FUNCTION_BLOCK FB_GenerateHeartBeat
VAR_INPUT
END_VAR
VAR_OUTPUT
	iHeartBeat		: UINT;
END_VAR
VAR
	tInterval		: TIME := T#500ms;
	tonInterval		: TON;
END_VAR


tonInterval(IN := TRUE,
			PT := tInterval,
			Q => );

IF (tonInterval.Q) THEN
	tonInterval(IN := FALSE);
	iHeartBeat := iHeartBeat + 1;
	IF (iHeartBeat > 100) THEN
		iHeartBeat := 0;
	END_IF
END_IF

PROPERTY PUBLIC P_tInterval : TIME
GET
P_tInterval := tInterval;
END_GET
SET
tInterval := P_tInterval;
END_SET
END_PROPERTY

END_FUNCTION_BLOCK

(* stored: Version 1.1.0.1, ProductVersion 3.1.4024.2
   POU FB_GenerateHeartBeat: Id {6bee6d55-d938-4fe0-9989-ca0e6bc441cc}, SpecialFunc None
   Property P_tInterval: Id {b5e1b68c-752d-4dc7-bed3-9a1c9fe2dab1}
   Get Get: Id {9d3127e5-f39a-4ae0-9057-df0978f5b7f9}
   Set Set: Id {75d2d995-ddeb-415c-8525-ba551e30ab7c} *)
